{attribute 'GeneratedUsingTerminal: EK1122-0000-0018'}
{attribute addProperty BoxType "EK1122-0000-0018"}
{attribute addProperty Id "Beckhoff_ER4xxxsub_EK1100EK1100_AB5A94672A_0001_ER4174_0002_0016ER4174_F6F08E1219A_0002_ER4174_0002_0019ER4174_F6F08E1219A_0003_ER4374_0002_0018ER4374_8019271A36A_0004_ER4374_0002_0019ER4374_8019271A36"}
{attribute addProperty CRC "3665413899"}
{attribute addProperty Size "112"}
TYPE Beckhoff_ER4xxxEK1122_DA79C70B EXTENDS EK1122_AB5A9467 :
STRUCT
	{attribute addProperty Name "Beckhoff_ER4xxxsub_EK1100"}
	{attribute addProperty PreviousPort "Beckhoff ER4xxxEK1122 : D"}
	Beckhoff_ER4xxxsub_EK1100 : EK1100_AB5A9467;
	{attribute addProperty Name "A_0001_ER4174_0002_0016"}
	{attribute addProperty PreviousPort "Beckhoff ER4xxxsub EK1100 : C"}
	A_0001_ER4174_0002_0016 : ER4174_F6F08E12;
	{attribute addProperty Name "A_0002_ER4174_0002_0019"}
	{attribute addProperty PreviousPort "A_0001(ER4174-0002-0016) : B"}
	A_0002_ER4174_0002_0019 : ER4174_F6F08E12;
	{attribute addProperty Name "A_0003_ER4374_0002_0018"}
	{attribute addProperty PreviousPort "A_0002(ER4174-0002-0019) : B"}
	A_0003_ER4374_0002_0018 : ER4374_8019271A;
	{attribute addProperty Name "A_0004_ER4374_0002_0019"}
	{attribute addProperty PreviousPort "A_0003(ER4374-0002-0018) : B"}
	A_0004_ER4374_0002_0019 : ER4374_8019271A;
END_STRUCT
END_TYPE

(* stored: Version 1.2.0.0, ProductVersion 3.1.4024.9
   DUT Beckhoff_ER4xxxEK1122_DA79C70B: Id {c9b48411-4d7d-4bf2-a4e2-83c2032a1112} *)
